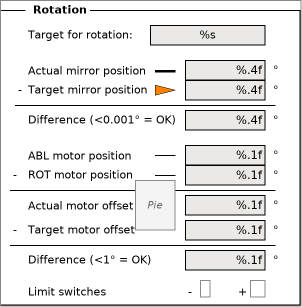
VISUALIZATION VISU_M3RotationDetails  // 302x307
VAR_IN_OUT
	ref : M3Rotation;
    widget : M3RotationWidget;
END_VAR
    Label (25,61 125x20), "Actual mirror position"
    Label (25,80 125x20), "Target mirror position"
    Line (0,10) (25,10)
    Label (30,0 150x20), "Rotation"
    Line (90,10) (300,10)
    Label (270,60 20x20), "°"
    Label (270,80 20x20), "°"
    Label (25,110 150x20), "Difference (<0.001° = OK)"
    Label (270,110 20x20), "°"
    Line (15,105) (275,105)
    Label (25,196 125x20), "Actual motor offset"
    Label (25,220 120x20), "Target motor offset"
    Label (270,195 20x20), "°"
    Label (270,220 20x20), "°"
    Label (25,250 130x20), "Difference (<1° = OK)"
    Label (270,250 20x20), "°"
    Line (10,245) (275,245)
    Rectangle (185,60 80x20), "%.4f", text variable: ref.actualPosition.degrees.value
    Rectangle (185,80 80x20), "%.4f", text variable: ref.target.position.degrees.value
    Rectangle (185,110 80x20), "%.4f", text variable: ref.actualPositionError.degrees.value
    Label (15,80 10x20), "-"
    Label (10,220 10x20), "-"
    Rectangle (185,195 80x20), "%.1f", text variable: ref.actualOffset.degrees.value
    Rectangle (185,220 80x20), "%.1f", text variable: ref.target.offset.degrees.value
    Rectangle (185,250 80x20), "%.1f", text variable: ref.actualOffsetError.degrees.value
    Polygon (175,90) (155,85) (155,95)
    Polygon (155,72) (155,70) (175,70) (175,72)
    Label (25,146 125x20), "ABL motor position"
    Label (270,145 20x20), "°"
    Label (270,165 20x20), "°"
    Line (10,190) (275,190)
    Label (10,165 10x20), "-"
    Rectangle (185,145 80x20), "%.1f", text variable: ref.parts.antiBacklashAxis.actPos.degrees.value
    Rectangle (185,165 80x20), "%.1f", text variable: ref.parts.positioningHallAxis.actPos.degrees.value
    Label (25,165 125x20), "ROT motor position"
    Rectangle (150,25 115x20), "%s", text variable: ref.target.actualStatus
    Pie (135,180 40x50)
    Line (155,175) (175,175)
    Line (155,155) (175,155)
    Label (25,25 125x20), "Target for rotation:"
    Label (25,282 130x20), "Limit switches"
    Label (185,282 15x20), "-"
    Frame (200,280 10x17)
        shows VISU_State_gray_red(state := ref.negativeLimitSwitchActive)
    Label (235,282 15x20), "+"
    Frame (250,280 15x17)
        shows VISU_State_gray_red(state := ref.positiveLimitSwitchActive)
    Line (0,305) (0,10)
    Line (300,305) (300,10)
    Line (300,305) (0,305)
END_VISUALIZATION

(* stored: Version 1.1.0.1, ProductVersion 3.1.4019.2
   Visu VISU_M3RotationDetails: Id {fcce902b-5e59-41d8-be5d-11398cd1ad17} *)
